# EPICS substitutions: apps/caenHvApp/Db/seq/richOnOff.substitutions
file "db/richOnOff.db" {
    pattern { DET ONOFF VAL }
    { RICH ON 1 }
    { RICH OFF 0 }
    { RICH2 ON 1 }
    { RICH2 OFF 0 }
}
